FUNCTION_BLOCK HandlingSequenceGoHome EXTENDS HandlingSequence IMPLEMENTS ZCore.ISequence
VAR
  _step : ZCore.Step(HandlingStep.GohomeBegin, HandlingStep.GohomeEnd);
  _timer : ZAux.Timer;
END_VAR

IF NOT Busy THEN
  RETURN;
END_IF

IF OnStart(_step) THEN
  ; // init custom sequence variables here ...
END_IF

IF OnStop() THEN
  RETURN; // external stop was triggered
END_IF

IF OnHalt() THEN
  ; // Halting := TRUE; // Uncomment to acknowledge that the sequence is halting
END_IF

REPEAT
  LogStep();

  CASE _step.Index OF
    (* -------------------------------------------------------------------------------------------------------------------------------- *)
    HandlingStep.GoHomeBegin:
    (* -------------------------------------------------------------------------------------------------------------------------------- *)
      IF _step.OnEntry()
      THEN
        _timer.WaitAsync(2);
			END_IF
      
      Await(_timer, nextStep:=HandlingStep.GoHomeEnd);
      // _step.SetNext(index:=HandlingStep.GoHomeEnd);

    (* -------------------------------------------------------------------------------------------------------------------------------- *)
    HandlingStep.GoHomeEnd:
    (* -------------------------------------------------------------------------------------------------------------------------------- *)
      SetBusy(FALSE);
  
  ELSE
    Abort('sequence contains unhandled step');
  END_CASE
UNTIL _step.IsNotRepeatable() OR_ELSE NOT Busy END_REPEAT

END_FUNCTION_BLOCK

(* stored: Version 1.1.0.1
   POU HandlingSequenceGoHome: Id {9cb9d926-3f0f-4e70-8efd-162f59776e7e}, SpecialFunc None *)
